// TIA Portal V18 export
TYPE "MEStoPLC_RecipeParameter_OP220"
// stored: IsFailsafeCompliant false
   STRUCT
      Press : "PresserRecipe";
      ATEQ { S7_SetPoint := 'True'} : "ATEQRecipe";
   END_STRUCT;
END_TYPE
